ABB RAPID module: Wobj_wobj_C2.mod

MODULE Wobj_wobj_C2
	! Points are read in order of declaration.
  ! Please do not change the order of points!

  LOCAL PERS robtarget pWobj_U_PointX1:=[[-1343.241,-1365.756,-669.9713],[0.00549515662714839,-0.69488924741745,-0.719045579433441,-0.00849862955510616],[-2,-1,-1,0],[0,9E+09,9E+09,9E+09,9E+09,9E+09]];
	LOCAL PERS robtarget pWobj_U_PointX2:=[[-1313.57,-2169.277,-673.7792],[0.00554911699146032,-0.690318822860718,-0.723434567451477,-0.00846166908740997],[-2,-1,-1,0],[0,9E+09,9E+09,9E+09,9E+09,9E+09]];
	LOCAL PERS robtarget pWobj_U_PointY1:=[[-712.2482,-2144.575,-676.9374],[0.00554848834872246,-0.690318644046783,-0.723434686660767,-0.00846292264759541],[-2,-1,-1,0],[0,9E+09,9E+09,9E+09,9E+09,9E+09]];

ENDMODULE
